// LS Electric XG5000 project: fdas
// PLC NewPLC
// module base 0 slot 0: 입출력 모듈:XBC-DR32H (DC 24V 입력, 릴레이 출력 32점)
// module base 0 slot 1: 위치결정 모듈:XBF-PD02A (위치결정 펄스(LD)출력형, 2축)
// module base 0 slot 2: 출력 모듈:XBE-TN/TP16A (트랜지스터 출력, 16점 (싱크출력/소스출력))

PROGRAM NewProgram (task: 스캔 프로그램)

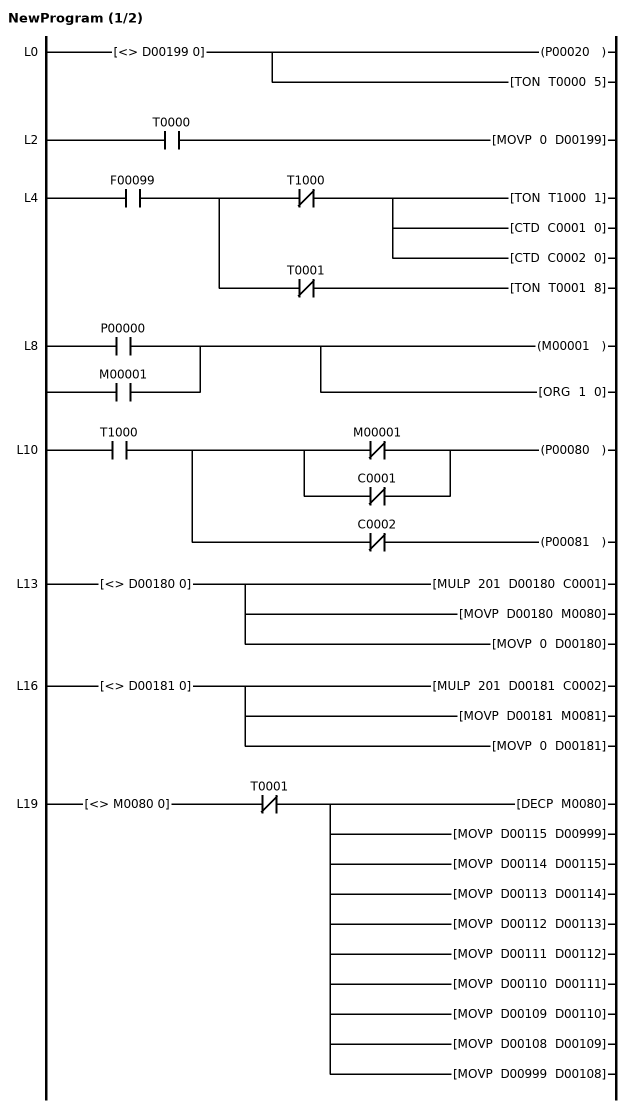
; L0
LOAD<>    D00199 0
OUT       P00020
TON       T0000 5
; L2
LOAD      T0000
MOVP      0 D00199
; L4
LOAD      F00099
MPUSH
AND NOT   T1000
TON       T1000 1
CTD       C0001 0
CTD       C0002 0
MPOP
AND NOT   T0001
TON       T0001 8
; L8
LOAD      P00000
OR        M00001
OUT       M00001
ORG       1 0
; L10
LOAD      T1000
MPUSH
LOAD NOT  M00001
OR NOT    C0001
AND LOAD
OUT       P00080
MPOP
AND NOT   C0002
OUT       P00081
; L13
LOAD<>    D00180 0
MULP      201 D00180 C0001
MOVP      D00180 M0080
MOVP      0 D00180
; L16
LOAD<>    D00181 0
MULP      201 D00181 C0002
MOVP      D00181 M0081
MOVP      0 D00181
; L19
LOAD<>    M0080 0
AND NOT   T0001
DECP      M0080
MOVP      D00115 D00999
MOVP      D00114 D00115
MOVP      D00113 D00114
MOVP      D00112 D00113
MOVP      D00111 D00112
MOVP      D00110 D00111
MOVP      D00109 D00110
MOVP      D00108 D00109
MOVP      D00999 D00108

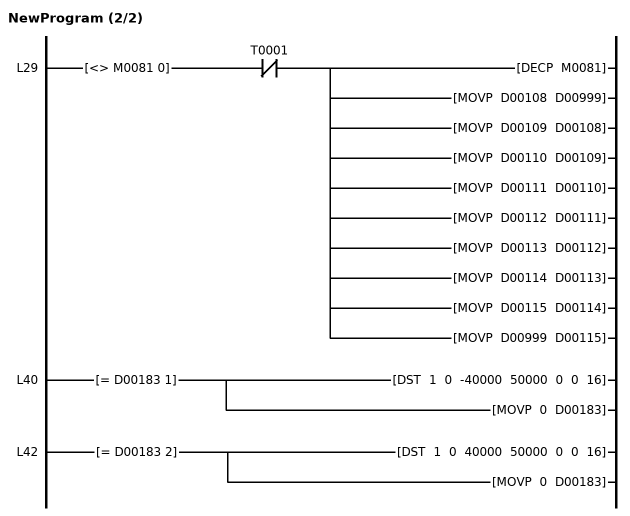
; L29
LOAD<>    M0081 0
AND NOT   T0001
DECP      M0081
MOVP      D00108 D00999
MOVP      D00109 D00108
MOVP      D00110 D00109
MOVP      D00111 D00110
MOVP      D00112 D00111
MOVP      D00113 D00112
MOVP      D00114 D00113
MOVP      D00115 D00114
MOVP      D00999 D00115
; L40
LOAD=     D00183 1
DST       1 0 -40000 50000 0 0 16
MOVP      0 D00183
; L42
LOAD=     D00183 2
DST       1 0 40000 50000 0 0 16
MOVP      0 D00183